TYPE
    TcoKeyMode_Config :
    STRUCT
        SwitKeyStanilisiation : TIME := T#500mS;

	
    END_STRUCT
END_TYPE

(* stored: Version 1.1.0.1
   DUT TcoKeyMode_Config: Id {e830eafc-2dd6-4e30-a3b3-05d8a78a12e0} *)
